{attribute 'linkalways'} 
{attribute 'no_explicit_call' := 'This FB is a CLASS and must be accessed using methods or properties'}
{attribute 'enable_dynamic_creation'}
FUNCTION_BLOCK FINAL LT_DWORD EXTENDS Node
VAR
	in1 : _DWORD(0);
	in2 : _DWORD(0);
	out : _BOOL(FALSE);
END_VAR

METHOD PUBLIC Clone : I_Node
VAR
	pNode : POINTER TO LT_DWORD;
END_VAR
pNode := __NEW(LT_DWORD);
Clone := pNode^;
END_METHOD

METHOD FB_init : BOOL
VAR_INPUT
	bInitRetains : BOOL; // if TRUE, the retain variables are initialized (warm start / cold start)
	bInCopyCode : BOOL;  // if TRUE, the instance afterwards gets moved into the copy code (online change)
END_VAR
AddInput('in1',THIS^.in1);
AddInput('in2',THIS^.in2);
AddOutput('out', THIS^.out);
END_METHOD

METHOD PROTECTED OnExecute
VAR
END_VAR
out.Value := in1.Value < in2.Value;
END_METHOD

END_FUNCTION_BLOCK

(* stored: Version 1.1.0.1, ProductVersion 3.1.4024.15
   POU LT_DWORD: Id {7856396f-a870-4770-a41d-72a0a1beba88}, SpecialFunc None
   Folder Constructor: Id {b547a3d7-d408-45ce-bd61-0c6f9d1c0d23}
   Method Clone: Id {d98e6cb6-9aa8-4c43-b704-8b21446236db}
   Method FB_init: Id {3474715d-8e40-4624-8d6d-dac3e458d3a0}
   Method OnExecute: Id {623ac237-5229-4d52-a7a1-936c72fb5692} *)
